// TIA Portal V19 export
TYPE "BTrk_item"
// stored: Access Published
   STRUCT
      B_ID : DInt;   // ID pezzo = trave = beam
      O_ID : DInt;   // ID ordine
      Quality : Int;   // Qualità: UNKNOW;GOOD;BAD...
      BLen_Meas : Real;   // Lunghezza pezzo misurata (dal pareggiatore)
      W_A : Real;   // Dim. base (W) = Altezza in impilamento (A)
      H_B : Real;   // Dim. altezza (H) = base in impilamento (B)
      P_L : Struct   // Dati Tracking della parte inferiore = Semi-Guscio
         P_ID : DInt;   // ID parte
         C_ID : DInt;   // ID rotolo
         Quality : Int;   // Qualità: UNKNOW;GOOD;BAD...
         PLen_Meas : Real;   // Lunghezza parte misurata (tra 2 tagli)
      END_STRUCT;
      P_U : Struct   // Dati Tracking della parte Superiore = Semi-Guscio
         P_ID : DInt;   // ID parte
         C_ID : DInt;   // ID rotolo
         Quality : Int;   // Qualità: UNKNOW;GOOD;BAD...
         PLen_Meas : Real;   // Lunghezza parte misurata (tra 2 tagli)
      END_STRUCT;
   END_STRUCT;
END_TYPE
